FUNCTION_BLOCK FB_BaseLoggerElementDecoratorParent IMPLEMENTS ITF_BaseLoggerElementDecoratorParent
VAR
	itfLoggerElement					: ITF_BaseLoggerElement;
END_VAR

(*			
	EVERDE sp. z o.o.
	Rafał Osajda		24.03.2025		TC 4024.66
	Definicja nowego zgłoszenia
*)
METHOD PUBLIC EventsDefinition : BOOL
EventsDefinition		:= THIS^.itfLoggerElement.EventsDefinition ();
END_METHOD

METHOD FB_init : BOOL
VAR_INPUT
	bInitRetains : BOOL; // if TRUE, the retain variables are initialized (warm start / cold start)
	bInCopyCode : BOOL;  // if TRUE, the instance afterwards gets moved into the copy code (online change)
	fbToDecorate		: ITF_DecoratedElement;
END_VAR
THIS^.itfLoggerElement	:= fbToDecorate.GetITFLoggerElement ();
END_METHOD

METHOD PUBLIC GetCode : STRING
VAR_INPUT
END_VAR
GetCode			:= THIS^.itfLoggerElement.GetCode ();
END_METHOD

METHOD PUBLIC GetID : UINT
VAR_INPUT
END_VAR
GetID		:= THIS^.GetID ();
END_METHOD

METHOD PUBLIC GetIdentyfier : ST_BaseElementIdentifier
VAR_INPUT
END_VAR
GetIdentyfier		:= THIS^.itfLoggerElement.GetIdentyfier ();
END_METHOD

METHOD PUBLIC GetName : ST_BaseLabel
VAR_INPUT
END_VAR
GetName		:= THIS^.itfLoggerElement.GetName ();
END_METHOD

METHOD PUBLIC GetType : E_BaseElementType
VAR_INPUT
END_VAR
GetType		:= THIS^.itfLoggerElement.GetType ();
END_METHOD

METHOD PUBLIC SetCode
VAR_INPUT
	sCode							: STRING;
	sAdd							: STRING;
END_VAR
THIS^.SetCode (sCode := sCode, sAdd := sAdd);
END_METHOD

(*			
	EVERDE sp. z o.o.
	Rafał Osajda		03.10.2025		TC 4024.66
	nadawanie unikalnych ID dla zdarzeń
*)
METHOD PUBLIC SetEventsIDs : UINT
VAR_INPUT
	uiNewID		: UINT;
END_VAR
SetEventsIDs		:= THIS^.itfLoggerElement.SetEventsIDs (uiNewID := uiNewID);
END_METHOD

METHOD PUBLIC SetID : UINT
VAR_INPUT
	uiID					: UINT;
END_VAR
SetID		:= THIS^.itfLoggerElement.SetID (uiID := uiID);
END_METHOD

METHOD PUBLIC SetName
VAR_INPUT
	stName				: ST_BaseLabel;
END_VAR
THIS^.itfLoggerElement.SetName (stName := stName);
END_METHOD

METHOD PUBLIC SetType
VAR_INPUT
	eType					: E_BaseElementType;
END_VAR
THIS^.SetType (eType := eType);
END_METHOD

END_FUNCTION_BLOCK

(* stored: Version 1.1.0.1, ProductVersion 3.1.4024.15
   POU FB_BaseLoggerElementDecoratorParent: Id {50e5d6fc-104d-4b44-8f8a-cca25a2c79ad}, SpecialFunc None
   Folder Events: Id {eb9e98c3-e9e7-4cc9-8f59-bda311616889}
   Folder ID: Id {9bc605ef-e9a8-4ca1-bc7f-dba9900e2bec}
   Method EventsDefinition: Id {ef9685f6-1abb-43a0-abc9-f3727e7f9f61}
   Method FB_init: Id {4e09a9fd-d946-4ab6-895c-bcd53dbd95e4}
   Method GetCode: Id {fb45a373-b3ec-477c-84f3-29c6ccc31846}
   Method GetID: Id {7145e0bd-f46a-4a46-805b-00dcaa8be6aa}
   Method GetIdentyfier: Id {ee5e55a7-e14a-4b70-9ae5-5db9318f2ede}
   Method GetName: Id {f7a38e19-aa17-4e41-a705-70b64f655ce3}
   Method GetType: Id {b3b491fe-5ca2-4dd8-92fa-7e2348d7e7e1}
   Method SetCode: Id {00b173e2-25bf-461c-8944-d24b4a8730d6}
   Method SetEventsIDs: Id {0dbdd410-7c26-4fe7-ada9-c4c6cde254d1}
   Method SetID: Id {d8abe519-9f2c-4cd9-b8c6-1023f5103b38}
   Method SetName: Id {59e013c8-0291-4059-a089-38561fa9d835}
   Method SetType: Id {990033cc-3aca-4d9d-83c5-feb482c0e6e8} *)
